// TIA Portal V17 export
// export: Created 2023-04-03T06:31:43.801568Z, ExportSetting WithDefaults, DisplayName Totally Integrated Automation Portal, DisplayVersion V17 Update 4, DisplayName TIA Portal Openness, DisplayVersion V17 Update 4, DisplayName TIA Portal Version Control Interface, DisplayVersion V17, DisplayName STEP 7 Professional, DisplayVersion V17 Update 4, DisplayName STEP 7 Safety, DisplayVersion V17, DisplayName WinCC Professional, DisplayVersion V17 Update 4
TYPE "SM"
// stored: IsFailsafeCompliant false
   STRUCT
      iSS1AssetSt : Int;
      iSS2AssetSt : Int;
      iSS1 : Int;
      iSS2 : Int;
   END_STRUCT;
END_TYPE
